ABB RobotStudio station: 4230.rsstn

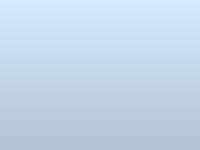
Station Station (saved by RobotStudio 6.7.7936.1011)
Layout (positions relative to the parent item):
  - Group_1 [graphiccomponentgroup]
  - IRB120_3_58__01_2 [mechanism, from Robots\IRB120_3_58_G_01.rslib] at (0, 0, 0) mm; joint values [0, 0, 0.0459, -0.1837, 0.0551, 0] (rad or m)
Targets, tools, work objects and paths stored in the station, written as RAPID:
! task T_ROB1
MODULE MTRN4230_Server_Sample
  PROC Main()
    MainServer;
  ENDPROC
  PROC CloseConnection()
  ENDPROC
  PROC MainServer()
    ListenForAndAcceptConnection;
    CloseConnection;
  ENDPROC
  PROC ListenForAndAcceptConnection()
  ENDPROC
ENDMODULE

! task T_ROB1
MODULE Assignment2
  PROC MainAss2()
    SingArea \Wrist;
    ConfJ \On;
    WaitTime 2;
    WaitTime 2;
    WaitTime 2;
    WaitTime 2;
  ENDPROC
ENDMODULE

